FUNCTION_BLOCK CmdAerate (* CAT Function Block Type *)
  (* Standard: 61499-2 *)
  (* Version 0.0, 6/7/2026, Schneider Electric, template *)
  PACKAGE SE.Nereda;
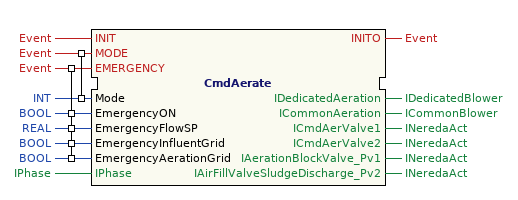
  EVENT_INPUT
    INIT;
    MODE WITH Mode;
    EMERGENCY WITH EmergencyON, EmergencyFlowSP, EmergencyInfluentGrid, EmergencyAerationGrid;
  END_EVENT
  EVENT_OUTPUT
    INITO;
  END_EVENT
  VAR_INPUT
    Mode : INT;
    EmergencyON : BOOL; (* Input event qualifier *)
    EmergencyFlowSP : REAL;
    EmergencyInfluentGrid : BOOL;
    EmergencyAerationGrid : BOOL;
  END_VAR
  SOCKETS
    IPhase : IPhase;
  END_SOCKETS
  PLUGS
    IDedicatedAeration : IDedicatedBlower;
    ICommonAeration : ICommonBlower;
  END_PLUGS
  PLUGS
    ICmdAerValve1 : INeredaAct;
    ICmdAerValve2 : INeredaAct;
    IAerationBlockValve_Pv1 : INeredaAct;
    IAirFillValveSludgeDischarge_Pv2 : INeredaAct;
  END_PLUGS
  (* 01 - FUNCTIONNAL INPUT INTERFACE *)
  (* 00 - INITIALIZATION *)
  (* 05 - LOGIC *)
  (* 06 - HMI INTERFACE *)
  (* 03 - FIELD INTERFACE *)
  (* 02 - FUNCTIONNAL OUTPUT INTERFACE *)
  (* Command Logic *)
  (* Capacity & Parameters Setpoint *)
  FBS
    IThis : CmdAerate_HMI(QI := TRUE);
    CmdLogic_DedicatedAeration : CmdDAerationValves; {SET_ATTRIBUTE(Configuration.Component.HideUnusedPorts, )}
    AerationInfluentGridParameterSelector : TowParametersSelector;
    AerationFlowSpSelector : ParametersSelector;
    CmdLogic_CommonAeration : CmdCAerationValves; {SET_ATTRIBUTE(Configuration.Component.HideUnusedPorts, )}
    DedicatedCommonSelector : CommonDedicatedSel;
  END_FBS
  EVENT_CONNECTIONS
    IPhase.Interlocked_CNF TO CmdLogic_DedicatedAeration.3B57434A9B977063;
    DedicatedCommonSelector.B6BCB327BF3D814B TO IPhase.REQ_Start_Ready;
    DedicatedCommonSelector.DFF9742BEF29F4B2 TO IPhase.REQ_Stop_Ready;
    DedicatedCommonSelector.E43C5E622E9EDB9D TO IPhase.REQ_Abort_Ready;
    MODE TO AerationInfluentGridParameterSelector.MODE;
    MODE TO AerationFlowSpSelector.MODE;
    EMERGENCY TO AerationFlowSpSelector.3B878B7E006C38E4;
    EMERGENCY TO AerationInfluentGridParameterSelector.3B878B7E006C38E4;
    AerationInfluentGridParameterSelector.CNF TO CmdLogic_DedicatedAeration.16F40D0A91C2944F;
    IDedicatedAeration.FB_BLOWER TO CmdLogic_DedicatedAeration.68A02AA49236F909;
    IDedicatedAeration.FB_BLOWER_AVAILABLE TO CmdLogic_DedicatedAeration.C5C063B1FA92898D;
    DedicatedCommonSelector.E6CE576DECE8FA36 TO IDedicatedAeration.START_BLOWER;
    AerationFlowSpSelector.CNF TO IDedicatedAeration.FLOW_SP_BLOWER;
    INIT TO IThis.C4758748B8B7D3EA;
    CmdLogic_CommonAeration.8657B668AE05B414 TO IThis.E235583F49B9570B;
    IThis.9FEA1874A72DD629 TO CmdLogic_DedicatedAeration.BD75C065B8FCDA05;
    IThis.AA5ACB8E8CB882BD TO AerationFlowSpSelector.REQ_NEREDA_VAL;
    IThis.3492549F473C0D4C TO AerationInfluentGridParameterSelector.REQ_NEREDA_VAL;
    IThis.B12E20154127E509 TO AerationInfluentGridParameterSelector.REQ_NEREDA_VAL;
    IThis.455769BEEFB660A8 TO AerationFlowSpSelector.REQ_MAN_VAL;
    IThis.1A8DF981889E9735 TO AerationInfluentGridParameterSelector.REQ_MAN_VAL;
    IThis.28D4F0947FCBA5C7 TO AerationInfluentGridParameterSelector.REQ_MAN_VAL;
    CmdLogic_CommonAeration.8657B668AE05B414 TO INITO;
    CmdLogic_DedicatedAeration.8657B668AE05B414 TO CmdLogic_CommonAeration.BD75C065B8FCDA05;
    IPhase.Interlocked_CNF TO CmdLogic_CommonAeration.3B57434A9B977063;
    CmdLogic_DedicatedAeration.84629170ACC8DE82 TO DedicatedCommonSelector.9CB3309E89E27687;
    CmdLogic_DedicatedAeration.BF1DFE7C21E469CA TO DedicatedCommonSelector.F2897017D62E0762;
    CmdLogic_DedicatedAeration.02F4D23CAC190EEC TO DedicatedCommonSelector.F758EF8250D0E827;
    CmdLogic_DedicatedAeration.7A769B3E526745F7 TO DedicatedCommonSelector.7C9DDB6CE58F5EAC;
    CmdLogic_CommonAeration.84629170ACC8DE82 TO DedicatedCommonSelector.9CB3309E89E27687;
    CmdLogic_CommonAeration.BF1DFE7C21E469CA TO DedicatedCommonSelector.F2897017D62E0762;
    CmdLogic_CommonAeration.02F4D23CAC190EEC TO DedicatedCommonSelector.F758EF8250D0E827;
    CmdLogic_CommonAeration.7A769B3E526745F7 TO DedicatedCommonSelector.7C9DDB6CE58F5EAC;
    IThis.DF194854A8102785 TO DedicatedCommonSelector.5CA6173F1C4E86FA;
    DedicatedCommonSelector.E6CE576DECE8FA36 TO ICommonAeration.START_BLOWER;
    AerationFlowSpSelector.CNF TO ICommonAeration.FLOW_SP_BLOWER;
    ICommonAeration.FB_BLOWER TO CmdLogic_CommonAeration.68A02AA49236F909;
    ICommonAeration.FB_BLOWER_AVAILABLE TO CmdLogic_CommonAeration.C5C063B1FA92898D;
  END_CONNECTIONS
  DATA_CONNECTIONS
    IPhase.Ready TO CmdLogic_DedicatedAeration.D9CFC7F0F0F8C6AB;
    IPhase.Starting TO CmdLogic_DedicatedAeration.40FB9C88801975DA;
    IPhase.Run TO CmdLogic_DedicatedAeration.61E0D6A9F4F73842;
    IPhase.Stopping TO CmdLogic_DedicatedAeration.C0695BB6BA34CA65;
    IPhase.Aborting TO CmdLogic_DedicatedAeration.4AD74DC94918733A;
    DedicatedCommonSelector.2A97C77077100C94 TO IPhase.Start_Ready;
    DedicatedCommonSelector.CA3438789A0EA1DF TO IPhase.Stop_Ready;
    DedicatedCommonSelector.0677B13F72D05C6B TO IPhase.Abort_Ready;
    Mode TO AerationInfluentGridParameterSelector.Mode;
    Mode TO AerationFlowSpSelector.Mode;
    EmergencyFlowSP TO AerationFlowSpSelector.4C6C1BFF70182CBB;
    EmergencyAerationGrid TO AerationInfluentGridParameterSelector.4C6C1BFF70182CBB;
    EmergencyInfluentGrid TO AerationInfluentGridParameterSelector.27A998BBD948DCC8;
    AerationInfluentGridParameterSelector.ValOut TO CmdLogic_DedicatedAeration.E6BA1C02D9C8B5E3;
    AerationInfluentGridParameterSelector.0957435043ED02C2 TO CmdLogic_DedicatedAeration.C182AB7746EC9FF3;
    IDedicatedAeration.FBStart TO CmdLogic_DedicatedAeration.D904E32D21E36958;
    IDedicatedAeration.FBStop TO CmdLogic_DedicatedAeration.58E8B9C3B04F91DA;
    IDedicatedAeration.FBBlowersAbailable TO CmdLogic_DedicatedAeration.F9BB5C3DA9C59D6E;
    DedicatedCommonSelector.1EF2595121C47467 TO IDedicatedAeration.StartBlower;
    AerationFlowSpSelector.ValOut TO IDedicatedAeration.FlowSPBlower;
    IThis.02BA975B3333A22E TO AerationFlowSpSelector.NeredaValue;
    IThis.307A045F4A4E620F TO AerationInfluentGridParameterSelector.NeredaValue;
    IThis.E67D4C76BBECB8AF TO AerationInfluentGridParameterSelector.A23B7BAC44D4E804;
    IThis.068083A73451FC27 TO AerationFlowSpSelector.ManValue;
    IThis.B51EE314AA8C1B45 TO AerationInfluentGridParameterSelector.ManValue;
    IThis.2E0B18D1C143649A TO AerationInfluentGridParameterSelector.90D08E776C3858FC;
    IPhase.Ready TO CmdLogic_CommonAeration.D9CFC7F0F0F8C6AB;
    IPhase.Starting TO CmdLogic_CommonAeration.40FB9C88801975DA;
    IPhase.Run TO CmdLogic_CommonAeration.61E0D6A9F4F73842;
    IPhase.Stopping TO CmdLogic_CommonAeration.C0695BB6BA34CA65;
    IPhase.Aborting TO CmdLogic_CommonAeration.4AD74DC94918733A;
    CmdLogic_DedicatedAeration.8BA48E88B36344BE TO DedicatedCommonSelector.4EABAE223D99E058;
    CmdLogic_DedicatedAeration.67F96BD12183C292 TO DedicatedCommonSelector.06E048E98F53EBF6;
    CmdLogic_DedicatedAeration.BD7F5AACD7869EC1 TO DedicatedCommonSelector.B02BDAA38C93975F;
    CmdLogic_DedicatedAeration.709CA1A54761FAAC TO DedicatedCommonSelector.D81231E47286A62F;
    CmdLogic_CommonAeration.8BA48E88B36344BE TO DedicatedCommonSelector.1F21147CB51C7EA6;
    CmdLogic_CommonAeration.67F96BD12183C292 TO DedicatedCommonSelector.EA1A5C22AD5895EC;
    CmdLogic_CommonAeration.BD7F5AACD7869EC1 TO DedicatedCommonSelector.6F7367F5CFF496A6;
    CmdLogic_CommonAeration.709CA1A54761FAAC TO DedicatedCommonSelector.D796844560BAB612;
    IThis.B143EF148481D958 TO DedicatedCommonSelector.6B7353E194B83739;
    DedicatedCommonSelector.1EF2595121C47467 TO ICommonAeration.StartBlower;
    AerationFlowSpSelector.ValOut TO ICommonAeration.FlowSPBlower;
    ICommonAeration.FBStart TO CmdLogic_CommonAeration.D904E32D21E36958;
    ICommonAeration.FBStop TO CmdLogic_CommonAeration.58E8B9C3B04F91DA;
    ICommonAeration.FBBlowersAbailable TO CmdLogic_CommonAeration.F9BB5C3DA9C59D6E;
  END_CONNECTIONS
  ADAPTER_CONNECTIONS
    CmdLogic_DedicatedAeration.452D64953B161AB4 TO ICmdAerValve1;
    CmdLogic_DedicatedAeration.6CE29B4C15302D9A TO ICmdAerValve2;
    CmdLogic_CommonAeration.0BC1BD7F7C60B585 TO IAerationBlockValve_Pv1;
    CmdLogic_CommonAeration.C7DB4697A0EA6C4A TO IAirFillValveSludgeDischarge_Pv2;
  END_CONNECTIONS
END_FUNCTION_BLOCK
